FUNCTION_BLOCK T_JogThroughStates EXTENDS T_UnitTestBase
VAR
  em : EquipmentModule;
  cmdTriggered : BOOL;
  actual, expected : Tc3_PackML_V2.E_PMLState;
  scanCounter : INT;
  myTestState : (ARRANGE, ACT, ASSERT);
END_VAR


CycleModuleLogicToAllowChangesToFilterThrough();

IF em.InitComplete THEN
  myTestState := ACT;
  em.ChangeState(E_PMLCommand.ePMLCommand_Clear);
END_IF

// clearing -> stopped
CycleModuleLogicToAllowChangesToFilterThrough();
actual := em.CurrentState;
assertion.AssertEquals_UINT(TO_UINT(actual), TO_UINT(E_PMLState.ePMLState_Stopped), 'clearing -> stopped assert : actual := em.CurrentState;');

// stopped -> Idle
em.ChangeState(E_PMLCommand.ePMLCommand_Reset);
CycleModuleLogicToAllowChangesToFilterThrough();
actual := em.CurrentState;
assertion.AssertEquals_UINT(TO_UINT(actual), TO_UINT(E_PMLState.ePMLState_Idle), 'stopped -> Idle assert : actual := em.CurrentState;');

// Idle - > Execute
em.ChangeState(E_PMLCommand.ePMLCommand_Start);
CycleModuleLogicToAllowChangesToFilterThrough();
actual := em.CurrentState;
assertion.AssertEquals_UINT(TO_UINT(actual), TO_UINT(E_PMLState.ePMLState_Execute), 'Idle - > Execute assert : actual := em.CurrentState;');

// Execute -> Hold
em.ChangeState(E_PMLCommand.ePMLCommand_Hold);
CycleModuleLogicToAllowChangesToFilterThrough();
actual := em.CurrentState;
assertion.AssertEquals_UINT(TO_UINT(actual), TO_UINT(E_PMLState.ePMLState_Held), 'Execute -> Hold assert : actual := em.CurrentState;');

// Hold -> Execute
em.ChangeState(E_PMLCommand.ePMLCommand_Unhold);
CycleModuleLogicToAllowChangesToFilterThrough();
actual := em.CurrentState;
assertion.AssertEquals_UINT(TO_UINT(actual), TO_UINT(E_PMLState.ePMLState_Execute), 'Hold -> Execute assert : actual := em.CurrentState;');

// Execute -> Suspend
em.ChangeState(E_PMLCommand.ePMLCommand_Suspend);
CycleModuleLogicToAllowChangesToFilterThrough();
actual := em.CurrentState;
assertion.AssertEquals_UINT(TO_UINT(actual), TO_UINT(E_PMLState.ePMLState_Suspended), 'Execute -> Suspend assert : actual := em.CurrentState;');

// Suspend - > Execute
em.ChangeState(E_PMLCommand.ePMLCommand_Unsuspend);
CycleModuleLogicToAllowChangesToFilterThrough();
actual := em.CurrentState;
assertion.AssertEquals_UINT(TO_UINT(actual), TO_UINT(E_PMLState.ePMLState_Execute), 'Suspend - > Execute assert : actual := em.CurrentState;');

// Execute -> Complete
em.ChangeState(E_PMLCommand.ePMLCommand_Complete);
CycleModuleLogicToAllowChangesToFilterThrough();
actual := em.CurrentState;
assertion.AssertEquals_UINT(TO_UINT(actual), TO_UINT(E_PMLState.ePMLState_Complete), 'Execute -> Complet assert : actual := em.CurrentState;');

// Complete -> Idle
em.ChangeState(E_PMLCommand.ePMLCommand_Reset);
CycleModuleLogicToAllowChangesToFilterThrough();
actual := em.CurrentState;
assertion.AssertEquals_UINT(TO_UINT(actual), TO_UINT(E_PMLState.ePMLState_Idle), 'Complete -> Idle assert : actual := em.CurrentState;');

// Idle -> Stopped
em.ChangeState(E_PMLCommand.ePMLCommand_Stop);
CycleModuleLogicToAllowChangesToFilterThrough();
actual := em.CurrentState;
assertion.AssertEquals_UINT(TO_UINT(actual), TO_UINT(E_PMLState.ePMLState_Stopped), 'Idle -> Stopped assert : actual := em.CurrentState;');

// Stopped -> Idle
em.ChangeState(E_PMLCommand.ePMLCommand_Reset);
CycleModuleLogicToAllowChangesToFilterThrough();
actual := em.CurrentState;
assertion.AssertEquals_UINT(TO_UINT(actual), TO_UINT(E_PMLState.ePMLState_Idle), 'Stopped -> Idle assert : actual := em.CurrentState;');

// Idle -> Abort
em.ChangeState(E_PMLCommand.ePMLCommand_Abort);
CycleModuleLogicToAllowChangesToFilterThrough();
actual := em.CurrentState;
assertion.AssertEquals_UINT(TO_UINT(actual), TO_UINT(E_PMLState.ePMLState_Aborted), 'Idle -> Abort assert : actual := em.CurrentState;');

TestFinished();

METHOD CycleModuleLogicToAllowChangesToFilterThrough : BOOL
VAR_INST
	i: INT;

END_VAR
//em.CyclicLogic();
//CycleModuleLogicToAllowChangesToFilterThrough := i >= 100;
//i := SEL(i >= 100, i + 1, 0);

FOR i := 0 TO 100 DO
  em.CyclicLogic();
END_FOR
END_METHOD

END_FUNCTION_BLOCK

(* stored: Version 1.1.0.1, ProductVersion 3.1.4024.12
   POU T_JogThroughStates: Id {2d0cac38-8dd5-4e55-9c85-df5389e732fb}, SpecialFunc None
   Method CycleModuleLogicToAllowChangesToFilterThrough: Id {c15eab2a-9e5a-4d0a-bd53-1f2df4e87a7c} *)
